// TwinCAT 3 PLC project Machine_Plc
// libraries:
//   Tc2_Standard, * (Beckhoff Automation GmbH)
// project tree:
//   / FB_Remote.TcPOU

// ---- FB_Remote.TcPOU

// :Description: Lives outside the solution directory; only reachable via the .sln reference.
FUNCTION_BLOCK FB_Remote
VAR
    counter : UDINT;
END_VAR


counter := counter + 1;

END_FUNCTION_BLOCK
